(* CODESYS project Trafikklys Biraveen.export

Project tree, tasks and I/O mapping:
  Device : CODESYS Control Win V3, 3S - Smart Software Solutions GmbH, version 3.5.16.30
    application Application
      libraries: Standard, * (System)
      task MainTask (cyclic, interval t#20ms, priority 1) calls PLC_PRG
      task VISU_TASK (cyclic, interval 100 ms, priority 31) calls VisuElems.Visu_Prg
      program PLC_PRG [CFC]
      function block trafikklys [ST]
      visualisation Visualization
*)

// Device/Application/PLC_PRG
PROGRAM PLC_PRG
VAR
	vektpad: BOOL;
	selvelyset: trafikklys;
	delay: TON;
END_VAR

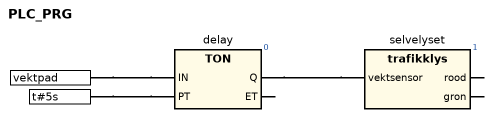
delay(IN := vektpad, PT := t#5s); // TON
selvelyset(vektsensor := delay.Q); // trafikklys

END_PROGRAM

// Device/Application/trafikklys
FUNCTION_BLOCK trafikklys
VAR_INPUT
		vektsensor: BOOL;
END_VAR
VAR_OUTPUT
	rood: BOOL;
	gron: BOOL;
END_VAR
VAR

END_VAR

IF vektsensor = TRUE THEN
	rood := FALSE;
	gron := TRUE;
END_IF


IF vektsensor = FALSE THEN
	rood := TRUE;
	gron := FALSE;
END_IF

END_FUNCTION_BLOCK

// Device/Application/Visualization
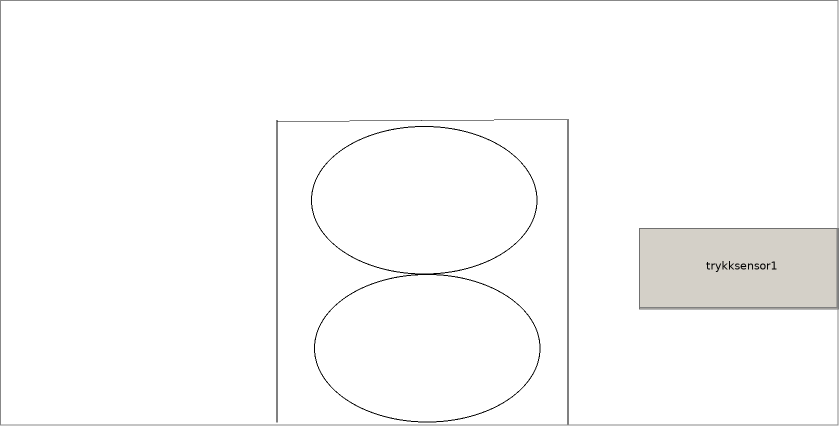
VISUALIZATION Visualization  // 839x426
    Line (277,422) (277,120)
    Line (565,425) (277,425)
    Line (568,424) (568,119)
    Line (277,121) (566,119)
    Ellipse (311,126 226x148)
        toggle PLC_PRG.selvelyset.rood
    Ellipse (314,274 226x148)
        toggle PLC_PRG.selvelyset.gron
    Button (639,228 200x81)
        toggle PLC_PRG.vektpad
    Label (667,251 150x30), "trykksensor1"
END_VISUALIZATION
